// TIA Portal V20 export
DATA_BLOCK "DB_Cognex"   // DB1255
// stored: AutoNumber false, InstanceOfName FB_Cognex, InstanceOfType FB
"FB_Cognex"
   // VAR
   //    sASTriggerReadyMemo : Bool;
   //    sASTriggerAckMemo : Bool;
   //    sASAcquiringMemo : Bool;
   //    sASMissedTrigMemo : Bool;
   //    sASOfflineResBit1Memo : Bool;
   //    sASOfflineResBit2Memo : Bool;
   //    sASOfflineResBit3Memo : Bool;
   //    sASOnlineMemo : Bool;
   //    sISInspectingMemo : Bool;
   //    sISToggleInspectDoneMemo : Bool;
   //    sISBufferOverrunMemo : Bool;
   //    sISResultsValidMemo : Bool;
   //    sISJobLoadingMemo : Bool;
   //    sISJobLoadCompleteMemo : Bool;
   //    sISJobLoadFailedMemo : Bool;
   //    sISSetUserDataACkMemo : Bool;
   //    sISJobPassMemo : Bool;
   //    sSEC0AckMemo : Bool;
   //    sSEC1AckMemo : Bool;
   //    sSEC2AckMemo : Bool;
   //    sSEC3AckMemo : Bool;
   //    sSEC4AckMemo : Bool;
   //    sSEC5AckMemo : Bool;
   //    sSEC6AckMemo : Bool;
   //    sSEC7AckMemo : Bool;
   //    sACTriggerEnableMemo : Bool;
   //    sACTriggerMemo : Bool;
   //    sACClearAcquirComplMemo : Bool;
   //    sACSetOfflineMemo : Bool;
   //    sICBufferResultsEnMemo : Bool;
   //    sICInspectResultsAckMemo : Bool;
   //    sICSetUserDataMemo : Bool;
   //    sICExecuteCmdMemo : Bool;
   //    sCCSetJobIDMemo : Int;
   //    sSEC0Memo : Bool;
   //    sSEC1Memo : Bool;
   //    sSEC2Memo : Bool;
   //    sSEC3Memo : Bool;
   //    sSEC4Memo : Bool;
   //    sSEC5Memo : Bool;
   //    sSEC6Memo : Bool;
   //    sSEC7Memo : Bool;
   //    sCamLightOn : Bool;
   //    sUserDataWrite : Bool;
   //    sUserDataWriteEn : Bool;
   //    sStartCapture : Bool;
   //    sAfterResultSoft7 : Bool;
   //    sTrigAckMemory : Bool;
   //    sMemoM55 : Bool;
   //    sSetSetup : Bool;
   //    sResultDataErrorBit : Bool;
   //    sICBufferResultsEnPositiveFront : Bool;
   //    sUserResultReadHole : Bool;
   //    sUserDataErrorBit : Bool;
   //    sIRActHoleNrResultMemo : Byte;
   //    sSetJobId : Int;
   //    sSetJobIdMemo : Int;
   //    sJCJobIDMemo : Word;
   //    sIRInspectionIDMemo : Word;
   //    sIRInspectResultCodeMemo : Word;
   //    sASAcquiNumMemo : Word;
   //    sUserDataErrorCode : Int;
   //    sResultDataErrorCode : Int;
   //    sNumChannel : Int;
   //    sCountAcquiNr : Int;
   //    sCounter : CTUD_INT;
   //    sUserDataArray : Array[0..7] of DWord;
   //    sResultDataArray : Array[0..3] of DWord;
   // END_VAR
BEGIN
END_DATA_BLOCK
